REGION Network 135: M333-FIXTURE 1 INTERNAL BLOWING SWITCH OFF / M56-SWITCH ON FIXTURE 2 INTERNAL BLOWING
   RUNG wire#powerrail
      Contact( "DB334_EXTENDED_M_CODE_UNIT_02_STA_0".M_code[333] )
      I_Contact( "DB356_M_UNIT_02_STA_0".M_CODES_UNIT_02_STA_0.Ack_M333 )
      I_Contact( "DB2120_MPP_ITC_IPC".RESET_FAULTS )
      I_Contact( "DB356_M_UNIT_02_STA_0".M_CODES_UNIT_02_STA_0.M_RESET_PULSE )
      Coil( "DB356_M_UNIT_02_STA_0".M_CODES_UNIT_02_STA_0.M333 )
   END_RUNG
   // the same network as SCL:
   "DB356_M_UNIT_02_STA_0".M_CODES_UNIT_02_STA_0.M333 := "DB334_EXTENDED_M_CODE_UNIT_02_STA_0".M_code[333] AND NOT "DB356_M_UNIT_02_STA_0".M_CODES_UNIT_02_STA_0.Ack_M333 AND NOT "DB2120_MPP_ITC_IPC".RESET_FAULTS AND NOT "DB356_M_UNIT_02_STA_0".M_CODES_UNIT_02_STA_0.M_RESET_PULSE;
END_REGION

REGION Network 136: ACKNOWLEDGE M334-FIXTURE 2 INTERNAL BLOWING SWITCH ON / ACKNOWLEDGE M57-SWITCH OFF FIXTURE 2 INTERNAL BLOWING
   RUNG wire#powerrail
      Contact( "DB356_M_UNIT_02_STA_0".M_CODES_UNIT_02_STA_0.M335 )
      Coil( "DB356_M_UNIT_02_STA_0".M_CODES_UNIT_02_STA_0.Ack_M334 )
   END_RUNG
   // the same network as SCL:
   "DB356_M_UNIT_02_STA_0".M_CODES_UNIT_02_STA_0.Ack_M334 := "DB356_M_UNIT_02_STA_0".M_CODES_UNIT_02_STA_0.M335;
END_REGION

REGION Network 137: M334-FIXTURE 2 INTERNAL BLOWING SWITCH ON / M57-SWITCH OFF FIXTURE 2 INTERNAL BLOWING
   RUNG wire#powerrail
      Contact( "DB334_EXTENDED_M_CODE_UNIT_02_STA_0".M_code[334] )
      wire#w1
      I_Contact( "DB356_M_UNIT_02_STA_0".M_CODES_UNIT_02_STA_0.Ack_M334 )
      I_Contact( "DB2120_MPP_ITC_IPC".RESET_FAULTS )
      I_Contact( "DB356_M_UNIT_02_STA_0".M_CODES_UNIT_02_STA_0.M_RESET_PULSE )
      Coil( "DB356_M_UNIT_02_STA_0".M_CODES_UNIT_02_STA_0.M334 )
   END_RUNG
   RUNG wire#powerrail
      Contact( "DB356_M_UNIT_02_STA_0".M_CODES_UNIT_02_STA_0.M334 )
   END_RUNG wire#w1
   // the same network as SCL:
   "DB356_M_UNIT_02_STA_0".M_CODES_UNIT_02_STA_0.M334 := ("DB334_EXTENDED_M_CODE_UNIT_02_STA_0".M_code[334] OR "DB356_M_UNIT_02_STA_0".M_CODES_UNIT_02_STA_0.M334) AND NOT "DB356_M_UNIT_02_STA_0".M_CODES_UNIT_02_STA_0.Ack_M334 AND NOT "DB2120_MPP_ITC_IPC".RESET_FAULTS AND NOT "DB356_M_UNIT_02_STA_0".M_CODES_UNIT_02_STA_0.M_RESET_PULSE;
END_REGION

REGION Network 138: ACKNOWLEDGE M335-FIXTURE 2 INTERNAL BLOWING SWITCH OFF
   RUNG wire#powerrail
      Contact( "M_ZERO" )
      Coil( "DB356_M_UNIT_02_STA_0".M_CODES_UNIT_02_STA_0.Ack_M335 )
   END_RUNG
   // the same network as SCL:
   "DB356_M_UNIT_02_STA_0".M_CODES_UNIT_02_STA_0.Ack_M335 := "M_ZERO";
END_REGION

REGION Network 139: M335-FIXTURE 2 INTERNAL BLOWING SWITCH OFF
   RUNG wire#powerrail
      Contact( "DB334_EXTENDED_M_CODE_UNIT_02_STA_0".M_code[335] )
      I_Contact( "DB356_M_UNIT_02_STA_0".M_CODES_UNIT_02_STA_0.Ack_M335 )
      I_Contact( "DB2120_MPP_ITC_IPC".RESET_FAULTS )
      I_Contact( "DB356_M_UNIT_02_STA_0".M_CODES_UNIT_02_STA_0.M_RESET_PULSE )
      Coil( "DB356_M_UNIT_02_STA_0".M_CODES_UNIT_02_STA_0.M335 )
   END_RUNG
   // the same network as SCL:
   "DB356_M_UNIT_02_STA_0".M_CODES_UNIT_02_STA_0.M335 := "DB334_EXTENDED_M_CODE_UNIT_02_STA_0".M_code[335] AND NOT "DB356_M_UNIT_02_STA_0".M_CODES_UNIT_02_STA_0.Ack_M335 AND NOT "DB2120_MPP_ITC_IPC".RESET_FAULTS AND NOT "DB356_M_UNIT_02_STA_0".M_CODES_UNIT_02_STA_0.M_RESET_PULSE;
END_REGION

REGION Network 140: READ-IN DISABLE / Read-in disable
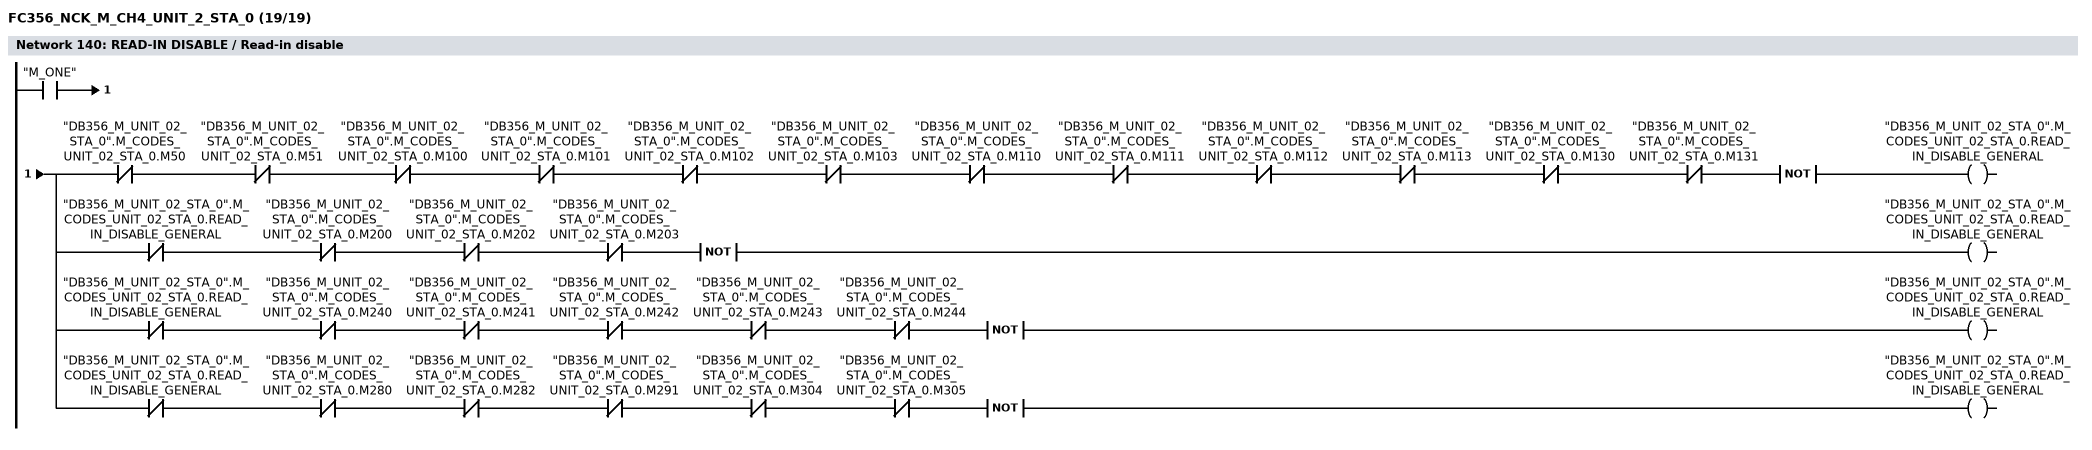
   RUNG wire#powerrail
      Contact( "M_ONE" )
      wire#w1
      I_Contact( "DB356_M_UNIT_02_STA_0".M_CODES_UNIT_02_STA_0.M50 )
      I_Contact( "DB356_M_UNIT_02_STA_0".M_CODES_UNIT_02_STA_0.M51 )
      I_Contact( "DB356_M_UNIT_02_STA_0".M_CODES_UNIT_02_STA_0.M100 )
      I_Contact( "DB356_M_UNIT_02_STA_0".M_CODES_UNIT_02_STA_0.M101 )
      I_Contact( "DB356_M_UNIT_02_STA_0".M_CODES_UNIT_02_STA_0.M102 )
      I_Contact( "DB356_M_UNIT_02_STA_0".M_CODES_UNIT_02_STA_0.M103 )
      I_Contact( "DB356_M_UNIT_02_STA_0".M_CODES_UNIT_02_STA_0.M110 )
      I_Contact( "DB356_M_UNIT_02_STA_0".M_CODES_UNIT_02_STA_0.M111 )
      I_Contact( "DB356_M_UNIT_02_STA_0".M_CODES_UNIT_02_STA_0.M112 )
      I_Contact( "DB356_M_UNIT_02_STA_0".M_CODES_UNIT_02_STA_0.M113 )
      I_Contact( "DB356_M_UNIT_02_STA_0".M_CODES_UNIT_02_STA_0.M130 )
      I_Contact( "DB356_M_UNIT_02_STA_0".M_CODES_UNIT_02_STA_0.M131 )
      Not()
      Coil( "DB356_M_UNIT_02_STA_0".M_CODES_UNIT_02_STA_0.READ_IN_DISABLE_GENERAL )
   END_RUNG
   RUNG wire#w1
      I_Contact( "DB356_M_UNIT_02_STA_0".M_CODES_UNIT_02_STA_0.READ_IN_DISABLE_GENERAL )
      I_Contact( "DB356_M_UNIT_02_STA_0".M_CODES_UNIT_02_STA_0.M200 )
      I_Contact( "DB356_M_UNIT_02_STA_0".M_CODES_UNIT_02_STA_0.M202 )
      I_Contact( "DB356_M_UNIT_02_STA_0".M_CODES_UNIT_02_STA_0.M203 )
      Not()
      Coil( "DB356_M_UNIT_02_STA_0".M_CODES_UNIT_02_STA_0.READ_IN_DISABLE_GENERAL )
   END_RUNG
   RUNG wire#w1
      I_Contact( "DB356_M_UNIT_02_STA_0".M_CODES_UNIT_02_STA_0.READ_IN_DISABLE_GENERAL )
      I_Contact( "DB356_M_UNIT_02_STA_0".M_CODES_UNIT_02_STA_0.M240 )
      I_Contact( "DB356_M_UNIT_02_STA_0".M_CODES_UNIT_02_STA_0.M241 )
      I_Contact( "DB356_M_UNIT_02_STA_0".M_CODES_UNIT_02_STA_0.M242 )
      I_Contact( "DB356_M_UNIT_02_STA_0".M_CODES_UNIT_02_STA_0.M243 )
      I_Contact( "DB356_M_UNIT_02_STA_0".M_CODES_UNIT_02_STA_0.M244 )
      Not()
      Coil( "DB356_M_UNIT_02_STA_0".M_CODES_UNIT_02_STA_0.READ_IN_DISABLE_GENERAL )
   END_RUNG
   RUNG wire#w1
      I_Contact( "DB356_M_UNIT_02_STA_0".M_CODES_UNIT_02_STA_0.READ_IN_DISABLE_GENERAL )
      I_Contact( "DB356_M_UNIT_02_STA_0".M_CODES_UNIT_02_STA_0.M280 )
      I_Contact( "DB356_M_UNIT_02_STA_0".M_CODES_UNIT_02_STA_0.M282 )
      I_Contact( "DB356_M_UNIT_02_STA_0".M_CODES_UNIT_02_STA_0.M291 )
      I_Contact( "DB356_M_UNIT_02_STA_0".M_CODES_UNIT_02_STA_0.M304 )
      I_Contact( "DB356_M_UNIT_02_STA_0".M_CODES_UNIT_02_STA_0.M305 )
      Not()
      Coil( "DB356_M_UNIT_02_STA_0".M_CODES_UNIT_02_STA_0.READ_IN_DISABLE_GENERAL )
   END_RUNG
   // the same network as SCL:
   "DB356_M_UNIT_02_STA_0".M_CODES_UNIT_02_STA_0.READ_IN_DISABLE_GENERAL := NOT ("M_ONE" AND NOT "DB356_M_UNIT_02_STA_0".M_CODES_UNIT_02_STA_0.M50 AND NOT "DB356_M_UNIT_02_STA_0".M_CODES_UNIT_02_STA_0.M51 AND NOT "DB356_M_UNIT_02_STA_0".M_CODES_UNIT_02_STA_0.M100 AND NOT "DB356_M_UNIT_02_STA_0".M_CODES_UNIT_02_STA_0.M101 AND NOT "DB356_M_UNIT_02_STA_0".M_CODES_UNIT_02_STA_0.M102 AND NOT "DB356_M_UNIT_02_STA_0".M_CODES_UNIT_02_STA_0.M103 AND NOT "DB356_M_UNIT_02_STA_0".M_CODES_UNIT_02_STA_0.M110 AND NOT "DB356_M_UNIT_02_STA_0".M_CODES_UNIT_02_STA_0.M111 AND NOT "DB356_M_UNIT_02_STA_0".M_CODES_UNIT_02_STA_0.M112 AND NOT "DB356_M_UNIT_02_STA_0".M_CODES_UNIT_02_STA_0.M113 AND NOT "DB356_M_UNIT_02_STA_0".M_CODES_UNIT_02_STA_0.M130 AND NOT "DB356_M_UNIT_02_STA_0".M_CODES_UNIT_02_STA_0.M131);
   "DB356_M_UNIT_02_STA_0".M_CODES_UNIT_02_STA_0.READ_IN_DISABLE_GENERAL := NOT ("M_ONE" AND NOT "DB356_M_UNIT_02_STA_0".M_CODES_UNIT_02_STA_0.READ_IN_DISABLE_GENERAL AND NOT "DB356_M_UNIT_02_STA_0".M_CODES_UNIT_02_STA_0.M200 AND NOT "DB356_M_UNIT_02_STA_0".M_CODES_UNIT_02_STA_0.M202 AND NOT "DB356_M_UNIT_02_STA_0".M_CODES_UNIT_02_STA_0.M203);
   "DB356_M_UNIT_02_STA_0".M_CODES_UNIT_02_STA_0.READ_IN_DISABLE_GENERAL := NOT ("M_ONE" AND NOT "DB356_M_UNIT_02_STA_0".M_CODES_UNIT_02_STA_0.READ_IN_DISABLE_GENERAL AND NOT "DB356_M_UNIT_02_STA_0".M_CODES_UNIT_02_STA_0.M240 AND NOT "DB356_M_UNIT_02_STA_0".M_CODES_UNIT_02_STA_0.M241 AND NOT "DB356_M_UNIT_02_STA_0".M_CODES_UNIT_02_STA_0.M242 AND NOT "DB356_M_UNIT_02_STA_0".M_CODES_UNIT_02_STA_0.M243 AND NOT "DB356_M_UNIT_02_STA_0".M_CODES_UNIT_02_STA_0.M244);
   "DB356_M_UNIT_02_STA_0".M_CODES_UNIT_02_STA_0.READ_IN_DISABLE_GENERAL := NOT ("M_ONE" AND NOT "DB356_M_UNIT_02_STA_0".M_CODES_UNIT_02_STA_0.READ_IN_DISABLE_GENERAL AND NOT "DB356_M_UNIT_02_STA_0".M_CODES_UNIT_02_STA_0.M280 AND NOT "DB356_M_UNIT_02_STA_0".M_CODES_UNIT_02_STA_0.M282 AND NOT "DB356_M_UNIT_02_STA_0".M_CODES_UNIT_02_STA_0.M291 AND NOT "DB356_M_UNIT_02_STA_0".M_CODES_UNIT_02_STA_0.M304 AND NOT "DB356_M_UNIT_02_STA_0".M_CODES_UNIT_02_STA_0.M305);
END_REGION
END_FUNCTION
